Staubli VAL3: avtomatskiCikel.pgx

program avtomatskiCikel()
begin

  // neskončna zanka pečenja palačink

  do
  //  call DodajMaso()
    //sDiag="Pečem prvo stran"
   // delay(nCas_peke1)
    //call obrat()
    //sDiag="Pečem drugo stran"
    //delay(nCas_peke2)
    //call naKroznik()
    call Glavni()
  until false
end
